// TIA Portal project "Programa_modelo_Github" (V16)

(* hardware
DEVICE "S71500/ET200MP station_1"  S7-1500 station
   slot 0: "Perfil soporte_0"  Rack  6ES7 590-1***0-0AA0
   slot 1: "PLC_1"  CPU 1516-3 PN/DP  6ES7 516-3AN01-0AB0  V2.8
      slot 3: "Display de la CPU_1"  6ES7591-1BA00-0AA0
      slot 32768: "Interfaz PROFINET_1"  X1
      slot 33024: "Interfaz PROFINET_2"  X2
      slot 33280: "Interfaz DP_1"  X3
      slot 34817: "Virtual CP interface port_1"  Virtual CP interface port  Virtual CP interface port
   slot 2: "DI 32x24VDC HF_1"  DI 32x24VDC HF  6ES7 521-1BL00-0AB0  V2.1
   slot 3: "DQ 32x24VDC/0.5A HF_1"  DQ 32x24VDC/0.5A HF  6ES7 522-1BL01-0AB0  V1.1
   slot 4: "AI 8xU/I/RTD/TC ST_1"  AI 8xU/I/RTD/TC ST  6ES7 531-7KF00-0AB0  V2.2
   slot 5: "AQ 4xU/I ST_1"  AQ 4xU/I ST  6ES7 532-5HD00-0AB0  V2.2
*)

// ===== PLC "PLC_1"  CPU 1516-3 PN/DP =====

VAR_GLOBAL   // PLC tag table "dos"
   "m1_do0" AT %Q0.0 : Bool;
   "m1_do1" AT %Q0.1 : Bool;
   "m1_do2" AT %Q0.2 : Bool;
   "m1_do3" AT %Q0.3 : Bool;
   "m1_do4" AT %Q0.4 : Bool;
   "m1_do5" AT %Q0.5 : Bool;
   "m1_do6" AT %Q0.6 : Bool;
   "m1_do7" AT %Q0.7 : Bool;
   "m1_do8" AT %Q1.0 : Bool;
   "m1_do9" AT %Q1.1 : Bool;
   "m1_do10" AT %Q1.2 : Bool;
   "m1_do11" AT %Q1.3 : Bool;
   "m1_do12" AT %Q1.4 : Bool;
   "m1_do13" AT %Q1.5 : Bool;
   "m1_do14" AT %Q1.6 : Bool;
   "m1_do15" AT %Q1.7 : Bool;
   "m1_do16" AT %Q2.0 : Bool;
   "m1_do17" AT %Q2.1 : Bool;
   "m1_do18" AT %Q2.2 : Bool;
   "m1_do19" AT %Q2.3 : Bool;
   "m1_do20" AT %Q2.4 : Bool;
   "m1_do21" AT %Q2.5 : Bool;
   "m1_do22" AT %Q2.6 : Bool;
   "m1_do23" AT %Q2.7 : Bool;
   "m1_do24" AT %Q3.0 : Bool;
   "m1_do25" AT %Q3.1 : Bool;
   "m1_do26" AT %Q3.2 : Bool;
   "m1_do27" AT %Q3.3 : Bool;
   "m1_do28" AT %Q3.4 : Bool;
   "m1_do29" AT %Q3.5 : Bool;
   "m1_do30" AT %Q3.6 : Bool;
   "m1_do31" AT %Q3.7 : Bool;
END_VAR

VAR_GLOBAL   // PLC tag table "dis"
   "m0_di0" AT %I0.0 : Bool;
   "m0_di1" AT %I0.1 : Bool;
   "m0_di2" AT %I0.2 : Bool;
   "m0_di3" AT %I0.3 : Bool;
   "m0_di4" AT %I0.4 : Bool;
   "m0_di5" AT %I0.5 : Bool;
   "m0_di6" AT %I0.6 : Bool;
   "m0_di7" AT %I0.7 : Bool;
   "m0_di8" AT %I1.0 : Bool;
   "m0_di9" AT %I1.1 : Bool;
   "m0_di10" AT %I1.2 : Bool;
   "m0_di11" AT %I1.3 : Bool;
   "m0_di12" AT %I1.4 : Bool;
   "m0_di13" AT %I1.5 : Bool;
   "m0_di14" AT %I1.6 : Bool;
   "m0_di15" AT %I1.7 : Bool;
   "m0_di16" AT %I2.0 : Bool;
   "m0_di17" AT %I2.1 : Bool;
   "m0_di18" AT %I2.2 : Bool;
   "m0_di19" AT %I2.3 : Bool;
   "m0_di20" AT %I2.4 : Bool;
   "m0_di21" AT %I2.5 : Bool;
   "m0_di22" AT %I2.6 : Bool;
   "m0_di23" AT %I2.7 : Bool;
   "m0_di24" AT %I3.0 : Bool;
   "m0_di25" AT %I3.1 : Bool;
   "m0_di26" AT %I3.2 : Bool;
   "m0_di27" AT %I3.3 : Bool;
   "m0_di28" AT %I3.4 : Bool;
   "m0_di29" AT %I3.5 : Bool;
   "m0_di30" AT %I3.6 : Bool;
END_VAR

TYPE "di_t"
   STRUCT
      start_button : Bool;
      stop_button : Bool;
      emergency_stop : Bool;
      reset_button : Bool;
      cylinder_position_down_2b1 : Bool;
      cylinder_position_up_2b2 : Bool;
      motor_begin_sensor_1b1 : Bool;
      motor_intermediate_sensor_1b3 : Bool;
      motor_final_sensor_1b2 : Bool;
      product_sensor_base_av1 : Bool;
      termic_protection : Bool;
      clamp_sensor_3b1 : Bool;
   END_STRUCT;
END_TYPE

TYPE "do_t"
   STRUCT
      motor_turn_left : Bool;
      motor_turn_right : Bool;
      cylinder_down : Bool;
      cylinder_up : Bool;
      clamp_open : Bool;
      clamp_close : Bool;
   END_STRUCT;
END_TYPE

TYPE "signals_t"
   STRUCT
      di : "di_t";
      "do" : "do_t";
      permisions : "do_t";
   END_STRUCT;
END_TYPE

DATA_BLOCK "gvar"   // DB1
{ S7_Optimized_Access := 'TRUE' }
VERSION : 0.1
   VAR
      summary_error : Bool;
      signals : "signals_t";
   END_VAR
BEGIN
END_DATA_BLOCK

ORGANIZATION_BLOCK "Main"   // OB1, LAD, ProgramCycle
TITLE = "Main Program Sweep (Cycle)"
{ S7_Optimized_Access := 'TRUE' }
VERSION : 0.1
   VAR_INPUT
      Initial_Call : Bool;   // Initial call of this OB
      Remanence : Bool;   // =True, if remanent data are available
   END_VAR
   VAR_TEMP   // added for the SCL form of the ladder/FBD networks
      _w1 : Bool;
   END_VAR
BEGIN

REGION Network 1 (SCL): read inputs
   // Asignación de inputs fisicas a las inputs virtuales
END_REGION

REGION Network 2: errors managament
   // Tratamiento de errores que provoquen un paro de programa
END_REGION

REGION Network 3: program logic
   // Logica de funcionamiento de programa
END_REGION

REGION Network 4: actions restrictions
   // -SUPONDREMOS QUE VISTO EL MOTOR DESDE ARRIBA, EL GIRO A IZQUIERDAS ES IR HACIA LAS CINTAS Y EL GIRO A DERECHAS SERA VOLVER AL INICIO.SE TENDRA QUE COMPROBAR IN SITU EN LA INSTALACION.
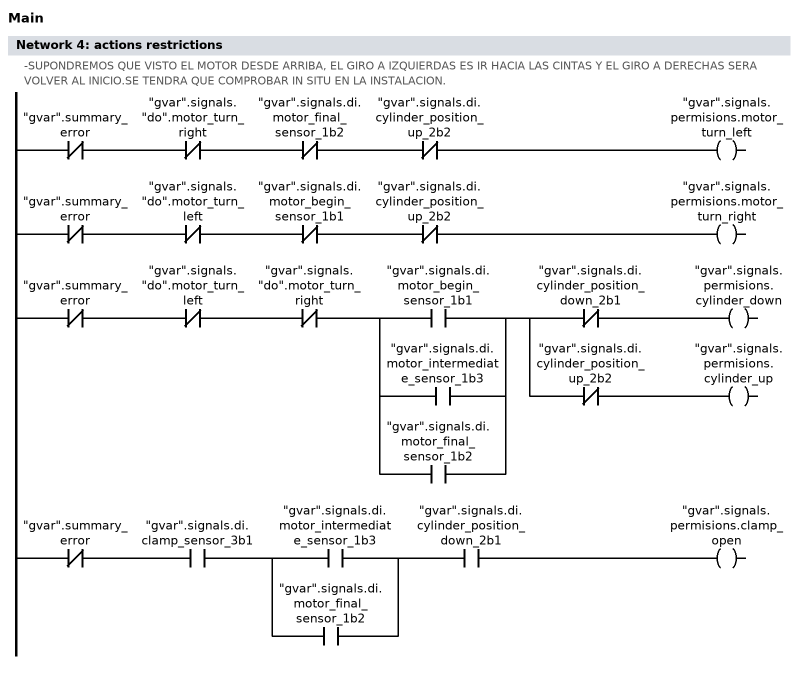
   RUNG wire#powerrail
      I_Contact( "gvar".summary_error )
      I_Contact( "gvar".signals."do".motor_turn_right )
      I_Contact( "gvar".signals.di.motor_final_sensor_1b2 )
      I_Contact( "gvar".signals.di.cylinder_position_up_2b2 )
      Coil( "gvar".signals.permisions.motor_turn_left )
   END_RUNG
   RUNG wire#powerrail
      I_Contact( "gvar".summary_error )
      I_Contact( "gvar".signals."do".motor_turn_left )
      I_Contact( "gvar".signals.di.motor_begin_sensor_1b1 )
      I_Contact( "gvar".signals.di.cylinder_position_up_2b2 )
      Coil( "gvar".signals.permisions.motor_turn_right )
   END_RUNG
   RUNG wire#powerrail
      I_Contact( "gvar".summary_error )
      I_Contact( "gvar".signals."do".motor_turn_left )
      I_Contact( "gvar".signals."do".motor_turn_right )
      wire#w1
      Contact( "gvar".signals.di.motor_begin_sensor_1b1 )
      wire#w2
      I_Contact( "gvar".signals.di.cylinder_position_down_2b1 )
      Coil( "gvar".signals.permisions.cylinder_down )
   END_RUNG
   RUNG wire#w1
      Contact( "gvar".signals.di.motor_intermediate_sensor_1b3 )
   END_RUNG wire#w2
   RUNG wire#w1
      Contact( "gvar".signals.di.motor_final_sensor_1b2 )
   END_RUNG wire#w2
   RUNG wire#w2
      I_Contact( "gvar".signals.di.cylinder_position_up_2b2 )
      Coil( "gvar".signals.permisions.cylinder_up )
   END_RUNG
   RUNG wire#powerrail
      I_Contact( "gvar".summary_error )
      Contact( "gvar".signals.di.clamp_sensor_3b1 )
      wire#w3
      Contact( "gvar".signals.di.motor_intermediate_sensor_1b3 )
      wire#w4
      Contact( "gvar".signals.di.cylinder_position_down_2b1 )
      Coil( "gvar".signals.permisions.clamp_open )
   END_RUNG
   RUNG wire#w3
      Contact( "gvar".signals.di.motor_final_sensor_1b2 )
   END_RUNG wire#w4
   // the same network as SCL:
   "gvar".signals.permisions.motor_turn_left := NOT "gvar".summary_error AND NOT "gvar".signals."do".motor_turn_right AND NOT "gvar".signals.di.motor_final_sensor_1b2 AND NOT "gvar".signals.di.cylinder_position_up_2b2;
   "gvar".signals.permisions.motor_turn_right := NOT "gvar".summary_error AND NOT "gvar".signals."do".motor_turn_left AND NOT "gvar".signals.di.motor_begin_sensor_1b1 AND NOT "gvar".signals.di.cylinder_position_up_2b2;
   #_w1 := NOT "gvar".summary_error AND NOT "gvar".signals."do".motor_turn_left AND NOT "gvar".signals."do".motor_turn_right AND ("gvar".signals.di.motor_begin_sensor_1b1 OR "gvar".signals.di.motor_intermediate_sensor_1b3 OR "gvar".signals.di.motor_final_sensor_1b2);
   "gvar".signals.permisions.cylinder_down := #_w1 AND NOT "gvar".signals.di.cylinder_position_down_2b1;
   "gvar".signals.permisions.cylinder_up := #_w1 AND NOT "gvar".signals.di.cylinder_position_up_2b2;
   "gvar".signals.permisions.clamp_open := NOT "gvar".summary_error AND "gvar".signals.di.clamp_sensor_3b1 AND ("gvar".signals.di.motor_intermediate_sensor_1b3 OR "gvar".signals.di.motor_final_sensor_1b2) AND "gvar".signals.di.cylinder_position_down_2b1;
END_REGION

REGION Network 5 (SCL): write inputs
   // Asignación de outputs virtuales a salidas reales
END_REGION
END_ORGANIZATION_BLOCK